(* IEC 61131-3 sources: eCockpitGit/test_project/src/%F%00 Library/%F%Common Functions/%F%String/%F%Normal/%F%Concat, 9 files *)

(* ---- %POU%FU_sConcat.st ---- *)
//This functions combines two strings
// |**Version**|**Author**| **Date** |**Changes**
// | 1         | NSN      | 13-06-18 | Creation
// | 1.1       | NSN      | 03-12-18 | Made pointers update in declaration
FUNCTION FU_sConcat : STRING(255)
VAR_INPUT
	s1			:STRING(255);			//Input String1
	s2			:STRING(255);			//Input String2
END_VAR
(*%!%__DELIMITER__%!%*)
FU_sConcatBIBO(sOut:=ADR(FU_sConcat),s1:=ADR(s1),s2:=ADR(s2),wOutSize:= 255);

(* ---- %POU%FU_sConcat10.st ---- *)
//This functions combines ten strings
// |**Version**|**Author**| **Date** |**Changes**
// | 1         | NSN      | 03-12-18 | Creation
FUNCTION FU_sConcat10 : STRING(255)
VAR_INPUT
	s1			:STRING(255);			//Input String1
	s2			:STRING(255);			//Input String2
	s3			:STRING(255);			//Input String3
	s4			:STRING(255);			//Input String4
	s5			:STRING(255);			//Input String5
	s6			:STRING(255);			//Input String6
	s7			:STRING(255);			//Input String7
	s8			:STRING(255);			//Input String8
	s9			:STRING(255);			//Input String9
	s10			:STRING(255);			//Input String10
END_VAR
(*%!%__DELIMITER__%!%*)
FU_sConcat10BIBO(sOut:=ADR(FU_sConcat10),s1:=ADR(s1),s2:=ADR(s2),s3:=ADR(s3),s4:=ADR(s4),s5:=ADR(s5),s6:=ADR(s6),s7:=ADR(s7),s8:=ADR(s8),s9:=ADR(s9),s10:=ADR(s10),wOutSize:=255);

(* ---- %POU%FU_sConcat3.st ---- *)
//This functions combines three strings
// |**Version**|**Author**| **Date** |**Changes**
// | 1         | NSN      | 03-12-18 | Creation
FUNCTION FU_sConcat3 : STRING(255)
VAR_INPUT
	s1			:STRING(255);			//Input String1
	s2			:STRING(255);			//Input String2
	s3			:STRING(255);			//Input String3
END_VAR
(*%!%__DELIMITER__%!%*)
FU_sConcat3BIBO(sOut:=ADR(FU_sConcat3),s1:=ADR(s1),s2:=ADR(s2),s3:=ADR(s3),wOutSize:=255);

(* ---- %POU%FU_sConcat4.st ---- *)
//This functions combines four strings
// |**Version**|**Author**| **Date** |**Changes**
// | 1         | NSN      | 03-12-18 | Creation
FUNCTION FU_sConcat4 : STRING(255)
VAR_INPUT
	s1			:STRING(255);			//Input String1
	s2			:STRING(255);			//Input String2
	s3			:STRING(255);			//Input String3
	s4			:STRING(255);			//Input String4
END_VAR
(*%!%__DELIMITER__%!%*)
FU_sConcat4BIBO(sOut:=ADR(FU_sConcat4),s1:=ADR(s1),s2:=ADR(s2),s3:=ADR(s3),s4:=ADR(s4),wOutSize:=255);

(* ---- %POU%FU_sConcat5.st ---- *)
//This functions combines five strings
// |**Version**|**Author**| **Date** |**Changes**
// | 1         | NSN      | 03-12-18 | Creation
FUNCTION FU_sConcat5 : STRING(255)
VAR_INPUT
	s1			:STRING(255);			//Input String1
	s2			:STRING(255);			//Input String2
	s3			:STRING(255);			//Input String3
	s4			:STRING(255);			//Input String4
	s5			:STRING(255);			//Input String5
END_VAR
(*%!%__DELIMITER__%!%*)
FU_sConcat5BIBO(sOut:=ADR(FU_sConcat5),s1:=ADR(s1),s2:=ADR(s2),s3:=ADR(s3),s4:=ADR(s4),s5:=ADR(s5),wOutSize:=255);

(* ---- %POU%FU_sConcat6.st ---- *)
//This functions combines six strings
// |**Version**|**Author**| **Date** |**Changes**
// | 1         | NSN      | 03-12-18 | Creation
FUNCTION FU_sConcat6 : STRING(255)
VAR_INPUT
	s1			:STRING(255);			//Input String1
	s2			:STRING(255);			//Input String2
	s3			:STRING(255);			//Input String3
	s4			:STRING(255);			//Input String4
	s5			:STRING(255);			//Input String5
	s6			:STRING(255);			//Input String6
END_VAR
(*%!%__DELIMITER__%!%*)
FU_sConcat6BIBO(sOut:=ADR(FU_sConcat6),s1:=ADR(s1),s2:=ADR(s2),s3:=ADR(s3),s4:=ADR(s4),s5:=ADR(s5),s6:=ADR(s6),wOutSize:=255);

(* ---- %POU%FU_sConcat7.st ---- *)
//This functions combines seven strings
// |**Version**|**Author**| **Date** |**Changes**
// | 1         | NSN      | 03-12-18 | Creation
FUNCTION FU_sConcat7 : STRING(255)
VAR_INPUT
	s1			:STRING(255);			//Input String1
	s2			:STRING(255);			//Input String2
	s3			:STRING(255);			//Input String3
	s4			:STRING(255);			//Input String4
	s5			:STRING(255);			//Input String5
	s6			:STRING(255);			//Input String6
	s7			:STRING(255);			//Input String7
END_VAR
(*%!%__DELIMITER__%!%*)
FU_sConcat7BIBO(sOut:=ADR(FU_sConcat7),s1:=ADR(s1),s2:=ADR(s2),s3:=ADR(s3),s4:=ADR(s4),s5:=ADR(s5),s6:=ADR(s6),s7:=ADR(s7),wOutSize:=255);

(* ---- %POU%FU_sConcat8.st ---- *)
//This functions combines nine strings
// |**Version**|**Author**| **Date** |**Changes**
// | 1         | NSN      | 03-12-18 | Creation
FUNCTION FU_sConcat8 : STRING(255)
VAR_INPUT
	s1			:STRING(255);			//Input String1
	s2			:STRING(255);			//Input String2
	s3			:STRING(255);			//Input String3
	s4			:STRING(255);			//Input String4
	s5			:STRING(255);			//Input String5
	s6			:STRING(255);			//Input String6
	s7			:STRING(255);			//Input String7
	s8			:STRING(255);			//Input String8
END_VAR

(*%!%__DELIMITER__%!%*)
FU_sConcat8BIBO(sOut:=ADR(FU_sConcat8),s1:=ADR(s1),s2:=ADR(s2),s3:=ADR(s3),s4:=ADR(s4),s5:=ADR(s5),s6:=ADR(s6),s7:=ADR(s7),s8:=ADR(s8),wOutSize:=255);

(* ---- %POU%FU_sConcat9.st ---- *)
//This functions combines nine strings
// |**Version**|**Author**| **Date** |**Changes**
// | 1         | NSN      | 03-12-18 | Creation
FUNCTION FU_sConcat9 : STRING(255)
VAR_INPUT
	s1			:STRING(255);			//Input String1
	s2			:STRING(255);			//Input String2
	s3			:STRING(255);			//Input String3
	s4			:STRING(255);			//Input String4
	s5			:STRING(255);			//Input String5
	s6			:STRING(255);			//Input String6
	s7			:STRING(255);			//Input String7
	s8			:STRING(255);			//Input String8
	s9			:STRING(255);			//Input String9
END_VAR
(*%!%__DELIMITER__%!%*)
FU_sConcat9BIBO(sOut:=ADR(FU_sConcat9),s1:=ADR(s1),s2:=ADR(s2),s3:=ADR(s3),s4:=ADR(s4),s5:=ADR(s5),s6:=ADR(s6),s7:=ADR(s7),s8:=ADR(s8),s9:=ADR(s9),wOutSize:=255);
